{attribute addProperty BoxType "EL3681-0000-0017"}
{attribute addProperty Id "CtrlAT %Q*Ctrl_D7097D21162"}
{attribute addProperty CRC "3819853773"}
{attribute addProperty SizeInBites "16"}
{attribute addProperty SizeInBytes "2"}
TYPE SAI_Range_E3AE57CD :
STRUCT
	{attribute addProperty Name "Ctrl"}
	Ctrl AT %Q* : Ctrl_D7097D21;
END_STRUCT
END_TYPE

(* stored: Version 1.2.0.0, ProductVersion 3.1.4024.9
   DUT SAI_Range_E3AE57CD: Id {a25bec7f-5826-4634-a3c7-ba67131519c3} *)
